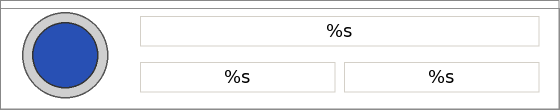
VISUALIZATION SingleSafeOutput_1  // 560x110
VAR_IN_OUT
	stDigitalOutput : ST_VisuCtrlOutputFrame;
END_VAR
    GroupBox (0,0 560x110)
        Lamp1 (15,5 100x100), variable: stDigitalOutput.bOut, style: Lamp-Lamp1-Blue
        Textfield (344,62 195x30), "%s", text variable: stDigitalOutput.sPortID
        Textfield (140,62 195x30), "%s", text variable: stDigitalOutput.sModuleType
        Textfield (140,16 399x30), "%s", text variable: stDigitalOutput.sName
END_VISUALIZATION

(* stored: Version 1.1.0.1, ProductVersion 3.1.4024.12
   Visu SingleSafeOutput_1: Id {cffb25b6-22e4-47db-a1e5-d42b454c5009} *)
